{attribute 'qualified_only'}
VAR_GLOBAL
	akt:					ST_ArtikelParameter;
END_VAR

(* stored: Version 1.1.0.1, ProductVersion 3.1.4024.12
   GVL ArtikelParam: Id {52f85db2-00b9-4516-81da-d3227ee72b00} *)
